PROGRAM POU_ALARM_120
VAR_INPUT
    xIN_QUIT      : BOOL; // Alarm quittieren
    iIN_ArraySize : INT;
    pstrIN_ALARM  : POINTER TO structAlarm;       // Array Alarmstruktur
    refPOU        : REFERENCE TO FB_AUT_ABSTRACT; // the POU to test
END_VAR
VAR_OUTPUT
    xOUT_AL_ST : BOOL; // Alarm Station aktiv
END_VAR
VAR
    //Alarmbaustein
    _FB_ALARM_ST : FB_ALARM;
    //Local
    iIndex : INT; // Index For Schleife	
END_VAR
VAR CONSTANT
    sDefString : STRING := 'Error ST120,'; // Station #
END_VAR

(********************** INITIALISIERE VARIABLEN ****************************)
FOR iIndex := 0 TO iIN_ArraySize - 1 DO
    pstrIN_ALARM[iIndex].xAlarmIN   := FALSE;
    pstrIN_ALARM[iIndex].xAlarmOFF  := FALSE;
    pstrIN_ALARM[iIndex].xAlarmSAVE := TRUE;
    pstrIN_ALARM[iIndex].xAlarmQUIT := xIN_QUIT;
    pstrIN_ALARM[iIndex].tAlarmVERZ := T#100MS;
    pstrIN_ALARM[iIndex].sAlarmText := '';
    pstrIN_ALARM[iIndex].bAlarmNr   := 0;
END_FOR

(********************** ALARME ****************************)
pstrIN_ALARM[0].xAlarmIN   := (refPOU.bOUT_ErrorNum = ST120_Alarm_e.Axis_120_01Y_error);
pstrIN_ALARM[0].sAlarmText := CONCAT(sDefString, ' Axis 01Y in error');
pstrIN_ALARM[0].bAlarmNr   := 0;

pstrIN_ALARM[1].xAlarmIN   := (refPOU.bOUT_ErrorNum = ST120_Alarm_e.Axis_120_02Z_error);
pstrIN_ALARM[1].sAlarmText := CONCAT(sDefString, ' Axis 02Z in error');
pstrIN_ALARM[1].bAlarmNr   := 0;

pstrIN_ALARM[2].xAlarmIN   := (refPOU.bOUT_ErrorNum = ST120_Alarm_e.Cylinder_griper_left);
pstrIN_ALARM[2].sAlarmText := CONCAT(sDefString, ' Cylinder .05 gripper right');
pstrIN_ALARM[2].bAlarmNr   := 0;

pstrIN_ALARM[3].xAlarmIN   := (refPOU.bOUT_ErrorNum = ST120_Alarm_e.Cylinder_griper_right);
pstrIN_ALARM[3].sAlarmText := CONCAT(sDefString, ' Cylinder .06 gripper left');
pstrIN_ALARM[3].bAlarmNr   := 0;

pstrIN_ALARM[4].xAlarmIN   := (refPOU.bOUT_ErrorNum = ST120_Alarm_e.Cylinder_pivot_left);
pstrIN_ALARM[4].sAlarmText := CONCAT(sDefString, ' Cylinder .06 pivot left');
pstrIN_ALARM[4].bAlarmNr   := 0;

pstrIN_ALARM[5].xAlarmIN   := (refPOU.bOUT_ErrorNum = ST120_Alarm_e.Cylinder_pivot_right);
pstrIN_ALARM[5].sAlarmText := CONCAT(sDefString, ' Cylinder .06 pivot left');
pstrIN_ALARM[5].bAlarmNr   := 0;

pstrIN_ALARM[6].xAlarmIN   := (refPOU.bOUT_ErrorNum = ST120_Alarm_e.Cylinder_hublader_left);
pstrIN_ALARM[6].sAlarmText := CONCAT(sDefString, ' Cylinder .06 hublader left');
pstrIN_ALARM[6].bAlarmNr   := 0;

pstrIN_ALARM[7].xAlarmIN   := (refPOU.bOUT_ErrorNum = ST120_Alarm_e.Cylinder_hublader_right);
pstrIN_ALARM[7].sAlarmText := CONCAT(sDefString, ' Cylinder .06 hublader left');
pstrIN_ALARM[7].bAlarmNr   := 0;

pstrIN_ALARM[8].xAlarmIN   := (refPOU.bOUT_ErrorNum = ST120_Alarm_e.Piece_in_unused_griper);
pstrIN_ALARM[8].sAlarmText := CONCAT(sDefString, ' One part is handled by a unused griper');
pstrIN_ALARM[8].bAlarmNr   := 0;

pstrIN_ALARM[9].xAlarmIN   := (refPOU.bOUT_ErrorNum = ST120_Alarm_e.Piece_missing_left_griper);
pstrIN_ALARM[9].sAlarmText := CONCAT(sDefString, ' A piece is missing in the left griper');
pstrIN_ALARM[9].bAlarmNr   := 0;

pstrIN_ALARM[10].xAlarmIN   := (refPOU.bOUT_ErrorNum = ST120_Alarm_e.Piece_missing_right_griper);
pstrIN_ALARM[10].sAlarmText := CONCAT(sDefString, ' A piece is missing in the right griper');
pstrIN_ALARM[10].bAlarmNr   := 0;

pstrIN_ALARM[11].xAlarmIN   := (refPOU.bOUT_ErrorNum = ST120_Alarm_e.Feeder_empty);
pstrIN_ALARM[11].sAlarmText := CONCAT(sDefString, ' The feeder is empty');
pstrIN_ALARM[11].bAlarmNr   := 0;

pstrIN_ALARM[12].xAlarmIN   := (refPOU.bOUT_ErrorNum = ST120_Alarm_e.Feeder_error);
pstrIN_ALARM[12].sAlarmText := CONCAT(sDefString, ' One part of the feeder is in error');
pstrIN_ALARM[12].bAlarmNr   := 0;

pstrIN_ALARM[13].xAlarmIN   := (refPOU.bOUT_ErrorNum = ST120_Alarm_e.Piece_in_unused_pivot);
pstrIN_ALARM[13].sAlarmText := CONCAT(sDefString, ' One part is handled by a unused pivot');
pstrIN_ALARM[13].bAlarmNr   := 0;

pstrIN_ALARM[14].xAlarmIN   := (refPOU.bOUT_ErrorNum = ST120_Alarm_e.Piece_missing_left_pivot);
pstrIN_ALARM[14].sAlarmText := CONCAT(sDefString, ' A piece is missing in the left pivot');
pstrIN_ALARM[14].bAlarmNr   := 0;

pstrIN_ALARM[15].xAlarmIN   := (refPOU.bOUT_ErrorNum = ST120_Alarm_e.Piece_missing_right_pivor);
pstrIN_ALARM[15].sAlarmText := CONCAT(sDefString, ' A piece is missing in the right pivot');
pstrIN_ALARM[15].bAlarmNr   := 0;

(********************** ALARM FB ****************************)
_FB_ALARM_ST(pstrIN_Alarm  := pstrIN_ALARM,
             iIN_ArraySize := ST120_Alarm_e._max);

(********************** ALARM FB ****************************)
xOUT_AL_ST := FALSE;

FOR iIndex := 0 TO iIN_ArraySize - 1 DO
    IF pstrIN_ALARM[iIndex].xAlarmOUT THEN
        xOUT_AL_ST := TRUE;
    END_IF
END_FOR

END_PROGRAM

(* stored: Version 1.1.0.1, ProductVersion 3.1.4024.6
   POU POU_ALARM_120: Id {0db29cbd-be82-4226-bf8c-f1f714b0ac1f}, SpecialFunc None *)
